KUKA KRL program: KVP_SendRelPos.src, KVP_SendRelPos.dat

--- KVP_SendRelPos.src ---
&ACCESS RVO
&REL 3
DEF KVP_SendRelPos( )

DECL E6AXIS HOME

MyRelBool = TRUE

BAS(#INITMOV,0)
BAS(#VEL_CP, 0.4)
BAS(#VEL_PTP, 20)
MyRelPos = $NULLFRAME
HOME = {E6AXIS: A1 90, A2 -90, A3 90, A4 0, A5 0, A6 0, E1 0, E2 0}

PTP HOME

WHILE MyRelBool
   PTP_REL MyRelPos
ENDWHILE

PTP HOME

END

--- KVP_SendRelPos.dat ---
&ACCESS RVO
&REL 3
DEFDAT KVP_SendRelPos PUBLIC

DECL E6POS MyRelPos
DECL BOOL MyRelBool

ENDDAT
